// SIMATIC S7-200 SMART project (STEP 7-Micro/WIN SMART), CPU ST40

SYMBOL_TABLE Table 1
Counter_1        C1
INIT_Done        M0.0
INIT_Error       MB1
SLAVE_Done       M0.1
SLAVE_Error      MB2
END_SYMBOL_TABLE

SYMBOL_TABLE System Symbols
Always_On        SM0.0    // Always ON
First_Scan_On    SM0.1    // ON for the first scan cycle only
Clock_1s         SM0.5    // Clock pulse that is ON for 0.5 s, OFF for 0.5 s, for a duty cycle time of 1 s.
END_SYMBOL_TABLE

ORGANIZATION_BLOCK MAIN:OB1
TITLE=Program Comments
BEGIN
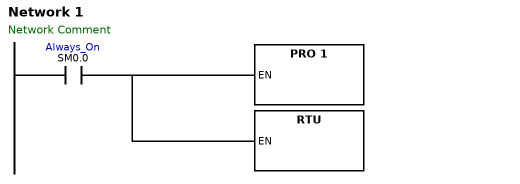
Network 1
// Network Comment
LD     Always_On:SM0.0
CALL   PRO 1:SBR10
CALL   RTU:SBR11
END_ORGANIZATION_BLOCK

// SBR0: protected block, not included

// SBR1: protected block, not included

// SBR2: protected block, not included

SUBROUTINE_BLOCK PRO 1:SBR10
TITLE=
BEGIN
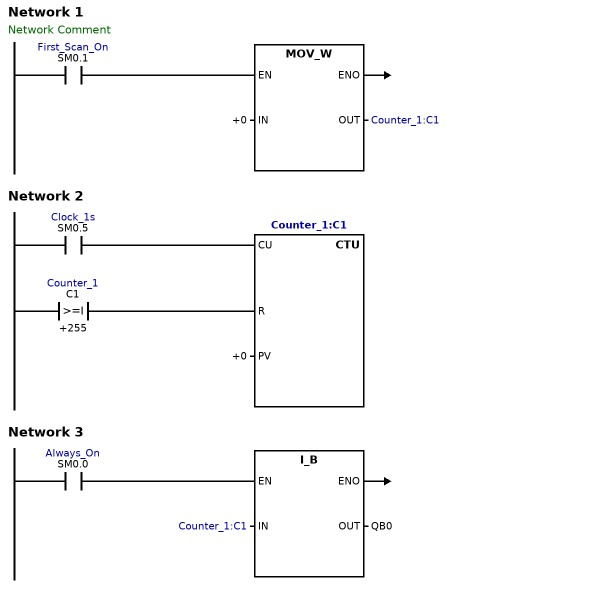
Network 1
// Network Comment
LD     First_Scan_On:SM0.1
MOVW   +0, Counter_1:C1
Network 2
LD     Clock_1s:SM0.5
LDW>=  Counter_1:C1, +255
CTU    Counter_1:C1, +0
Network 3
LD     Always_On:SM0.0
ITB    Counter_1:C1, QB0
END_SUBROUTINE_BLOCK

SUBROUTINE_BLOCK RTU:SBR11
TITLE=Subroutine Comments
BEGIN
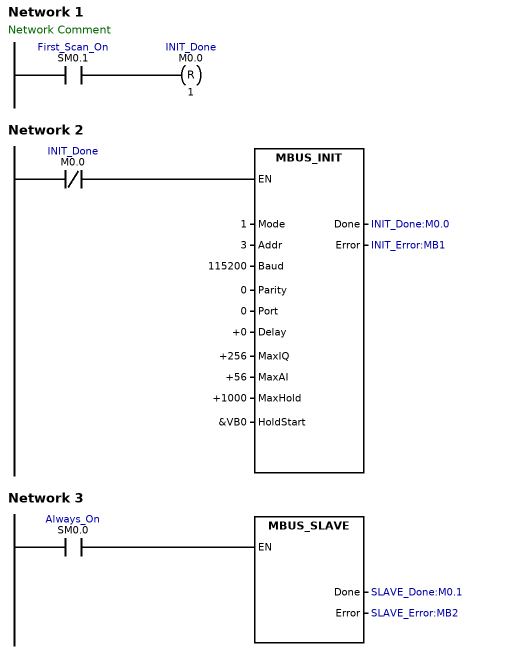
Network 1
// Network Comment
LD     First_Scan_On:SM0.1
R      INIT_Done:M0.0, 1
Network 2
LDN    INIT_Done:M0.0
CALL   MBUS_INIT:SBR0, 1, 3, 115200, 0, 0, +0, +256, +56, +1000, &VB0, INIT_Done:M0.0, INIT_Error:MB1
Network 3
LD     Always_On:SM0.0
CALL   MBUS_SLAVE:SBR1, SLAVE_Done:M0.1, SLAVE_Error:MB2
END_SUBROUTINE_BLOCK
